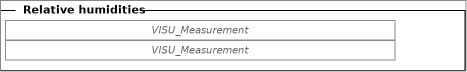
VISUALIZATION VISU_TelemetryRelativeHumidities  // 467x72
VAR_IN_OUT
    ref : TelemetryRelativeHumidities;
	widget : TelemetryRelativeHumiditiesWidget;
END_VAR
    Label (20,0 115x20), "Relative humidities"
    Line (465,70) (465,10)
        p2175578022: widget.actualStatus.color.bg
    Frame (5,20 390x20)
        shows VISU_Measurement(widget := widget.topAir)
    Frame (5,40 390x20)
        shows VISU_Measurement(widget := widget.insideTube)
    Line (140,10) (465,10)
        p2175578022: widget.actualStatus.color.bg
    Line (0,10) (15,10)
        p2175578022: widget.actualStatus.color.bg
    Line (0,70) (0,10)
        p2175578022: widget.actualStatus.color.bg
    Line (0,70) (465,70)
        p2175578022: widget.actualStatus.color.bg
END_VISUALIZATION

(* stored: Version 1.1.0.1, ProductVersion 3.1.4019.2
   Visu VISU_TelemetryRelativeHumidities: Id {4b95779e-9efb-4749-b85c-a679e7cc52bd} *)
